FUNCTION_BLOCK FB_Clock
VAR_INPUT
END_VAR
VAR_OUTPUT
END_VAR
VAR
END_VAR

END_FUNCTION_BLOCK

(* stored: Version 1.1.0.1, ProductVersion 3.1.4024.12
   POU FB_Clock: Id {0e267069-a3c3-4596-8c75-7a01d200315b}, SpecialFunc None *)
